// TIA Portal V16 program export: 1 tag tables, 0 data types, 1 data blocks, 4 code blocks (in call order from the OBs), 2 instance data blocks

VAR_GLOBAL   // PLC tag table "Default tag table"
   X_input AT %M0.0 : Bool;
   X_output AT %M0.1 : Bool;
END_VAR

DATA_BLOCK "Data_block_1"   // DB2
{ S7_Optimized_Access := 'TRUE' }
VERSION : 0.1
// stored: AutoNumber true, DBAccessibleFromOPCUA true, IsOnlyStoredInLoadMemory false, IsRetainMemResEnabled false, IsWriteProtectedInAS false, MemoryReserve 0
   VAR
      x : Bool;
      y : Bool;
      z : Bool;
      fc1_edge : Bool;
      fc1_catch_signal : Bool;
      fc1_output : Bool;
      "a" : Int;
      "b" : Int;
      c : Int;
      d : Int;
   END_VAR
BEGIN
END_DATA_BLOCK

ORGANIZATION_BLOCK "Main"   // OB1, LAD, ProgramCycle
TITLE = "Main Program Sweep (Cycle)"
{ S7_Optimized_Access := 'TRUE' }
VERSION : 0.1
// stored: AutoNumber true, IsIECCheckEnabled false, SetENOAutomatically false
   VAR_INPUT
      Initial_Call : Bool;   // Initial call of this OB
      Remanence : Bool;   // =True, if remanent data are available
   END_VAR
BEGIN

REGION Network 1
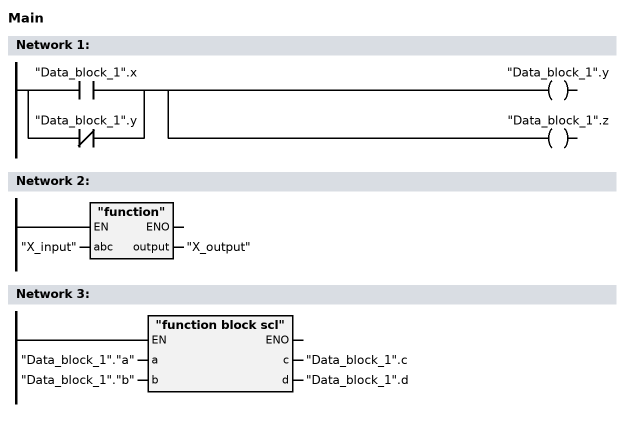
   RUNG wire#powerrail
      Contact( "Data_block_1".x )
      wire#w1
      Coil( "Data_block_1".y )
   END_RUNG
   RUNG wire#powerrail
      I_Contact( "Data_block_1".y )
   END_RUNG wire#w1
   RUNG wire#w1
      Coil( "Data_block_1".z )
   END_RUNG
   // the same network as SCL:
   "Data_block_1".y := "Data_block_1".x OR NOT "Data_block_1".y;
   "Data_block_1".z := "Data_block_1".y;
END_REGION

REGION Network 2
   RUNG wire#powerrail
      "function"(abc := "X_input", output => "X_output")
   END_RUNG
   // the same network as SCL:
   "function"(abc := "X_input", output => "X_output");
END_REGION

REGION Network 3
   RUNG wire#powerrail
      "function block scl"("a" := "Data_block_1"."a", "b" := "Data_block_1"."b", c => "Data_block_1".c, d => "Data_block_1".d)
   END_RUNG
   // the same network as SCL:
   "function block scl"("a" := "Data_block_1"."a",
                        "b" := "Data_block_1"."b",
                        c => "Data_block_1".c,
                        d => "Data_block_1".d);
END_REGION
END_ORGANIZATION_BLOCK

FUNCTION "function" : Void   // FC1, LAD
{ S7_Optimized_Access := 'TRUE' }
VERSION : 0.1
// stored: AutoNumber true, IsIECCheckEnabled false, SetENOAutomatically false, UDAEnableTagReadback false
   VAR_INPUT
      abc : Bool;
   END_VAR
   VAR_OUTPUT
      output : Bool;
   END_VAR
   VAR_TEMP
      intermediate : Bool;
   END_VAR
   VAR_TEMP   // added for the SCL form of the ladder/FBD networks
      _w1 : Bool;
   END_VAR
BEGIN

REGION Network 1
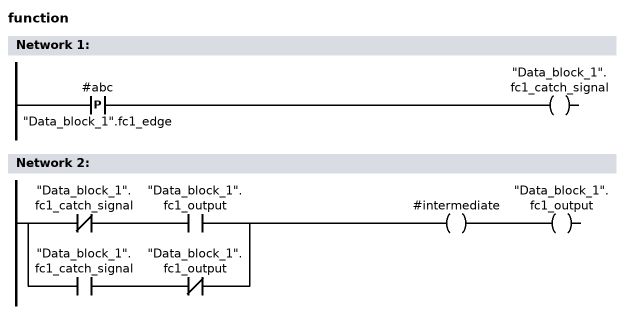
   RUNG wire#powerrail
      P_Contact(operand := #abc, bit := "Data_block_1".fc1_edge)
      Coil( "Data_block_1".fc1_catch_signal )
   END_RUNG
   // the same network as SCL:
   #_w1 := #abc AND NOT "Data_block_1".fc1_edge;   // rising edge of #abc
   "Data_block_1".fc1_edge := #abc;
   "Data_block_1".fc1_catch_signal := #_w1;
END_REGION

REGION Network 2
   RUNG wire#powerrail
      I_Contact( "Data_block_1".fc1_catch_signal )
      Contact( "Data_block_1".fc1_output )
      wire#w1
      Coil( #intermediate )
      Coil( "Data_block_1".fc1_output )
   END_RUNG
   RUNG wire#powerrail
      Contact( "Data_block_1".fc1_catch_signal )
      I_Contact( "Data_block_1".fc1_output )
   END_RUNG wire#w1
   // the same network as SCL:
   #intermediate := (NOT "Data_block_1".fc1_catch_signal AND "Data_block_1".fc1_output) OR ("Data_block_1".fc1_catch_signal AND NOT "Data_block_1".fc1_output);
   "Data_block_1".fc1_output := #intermediate;
END_REGION
END_FUNCTION

FUNCTION "function block scl" : Void
{ S7_Optimized_Access := 'TRUE' }
VERSION : 0.1
   VAR_INPUT 
      a : Int;
      b : Int;
   END_VAR

   VAR_OUTPUT 
      c : Int;
      d : Int;
   END_VAR


BEGIN
	//was is das
	#c := #a + #b;
	#d := #b - #c;
END_FUNCTION

FUNCTION_BLOCK "Main_Safety_RTG1"   // FB1, F_FBD
{ S7_Optimized_Access := 'TRUE' }
VERSION : 0.1
// stored: AutoNumber false, IsIECCheckEnabled false, UDAEnableTagReadback false
BEGIN
END_FUNCTION_BLOCK

DATA_BLOCK "Main_Safety_RTG1_DB"   // DB1, F_DB
NAME : FUSI
VERSION : 0.1
// stored: AutoNumber true, DBAccessibleFromOPCUA true, InstanceOfName Main_Safety_RTG1, InstanceOfType FB
"Main_Safety_RTG1"
BEGIN
END_DATA_BLOCK

DATA_BLOCK "function block scl_DB"   // DB3
VERSION : 0.1
// stored: AutoNumber true, DBAccessibleFromOPCUA true, InstanceOfName function block scl, InstanceOfType FB
"function block scl"
BEGIN
END_DATA_BLOCK
